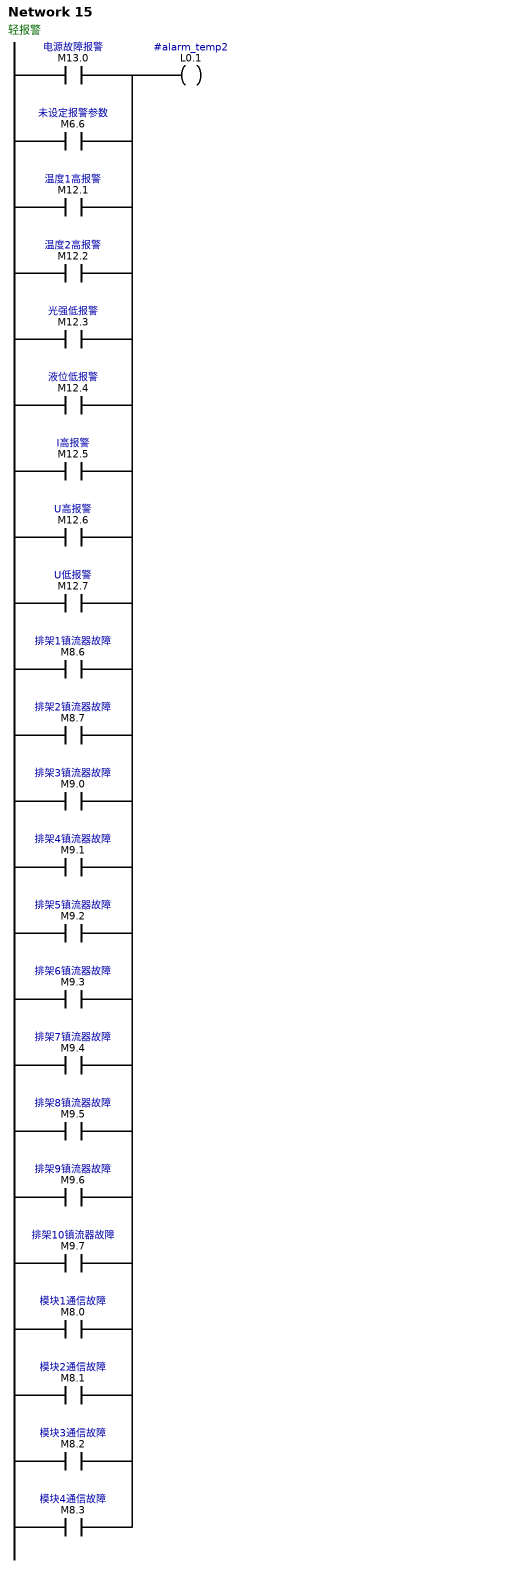
[picture p24: SBR7 networks 15-15]
Network 15
// 轻报警
LD     电源故障报警:M13.0
O      未设定报警参数:M6.6
O      温度1高报警:M12.1
O      温度2高报警:M12.2
O      光强低报警:M12.3
O      液位低报警:M12.4
O      I高报警:M12.5
O      U高报警:M12.6
O      U低报警:M12.7
O      排架1镇流器故障:M8.6
O      排架2镇流器故障:M8.7
O      排架3镇流器故障:M9.0
O      排架4镇流器故障:M9.1
O      排架5镇流器故障:M9.2
O      排架6镇流器故障:M9.3
O      排架7镇流器故障:M9.4
O      排架8镇流器故障:M9.5
O      排架9镇流器故障:M9.6
O      排架10镇流器故障:M9.7
O      模块1通信故障:M8.0
O      模块2通信故障:M8.1
O      模块3通信故障:M8.2
O      模块4通信故障:M8.3
=      #alarm_temp2:L0.1
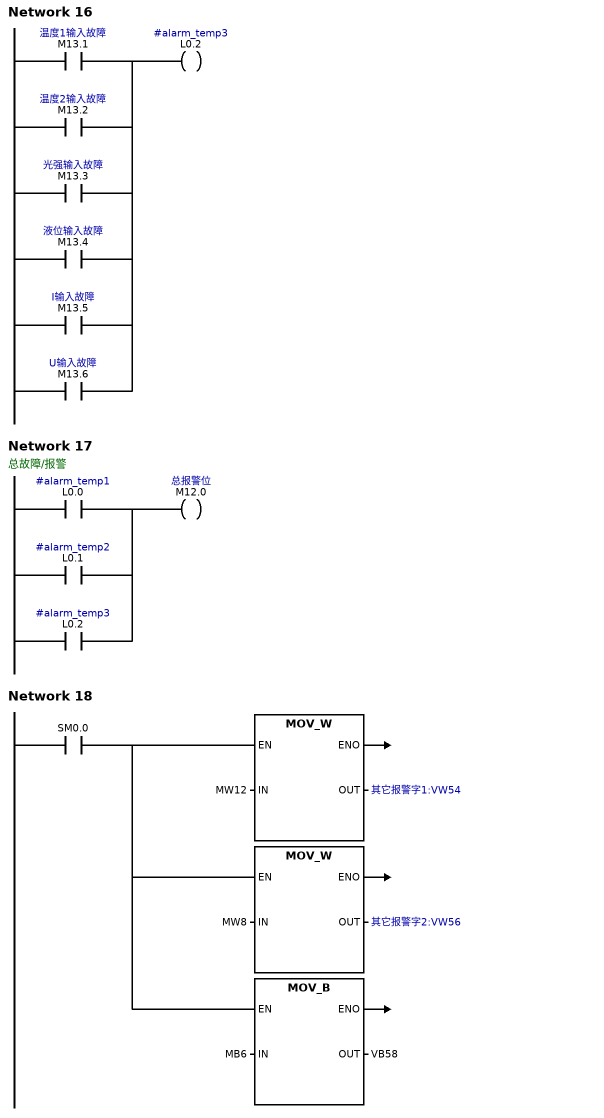
Network 16
LD     温度1输入故障:M13.1
O      温度2输入故障:M13.2
O      光强输入故障:M13.3
O      液位输入故障:M13.4
O      I输入故障:M13.5
O      U输入故障:M13.6
=      #alarm_temp3:L0.2
Network 17
// 总故障/报警
LD     #alarm_temp1:L0.0
O      #alarm_temp2:L0.1
O      #alarm_temp3:L0.2
=      总报警位:M12.0
Network 18
LD     SM0.0
MOVW   MW12, 其它报警字1:VW54
MOVW   MW8, 其它报警字2:VW56
MOVB   MB6, VB58
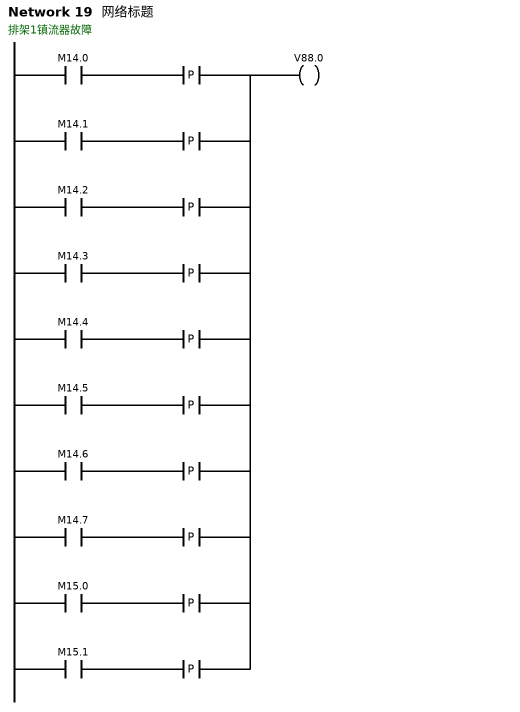
Network 19 // 网络标题
// 排架1镇流器故障
LD     M14.0
EU
LD     M14.1
EU
OLD
LD     M14.2
EU
OLD
LD     M14.3
EU
OLD
LD     M14.4
EU
OLD
LD     M14.5
EU
OLD
LD     M14.6
EU
OLD
LD     M14.7
EU
OLD
LD     M15.0
EU
OLD
LD     M15.1
EU
OLD
=      V88.0
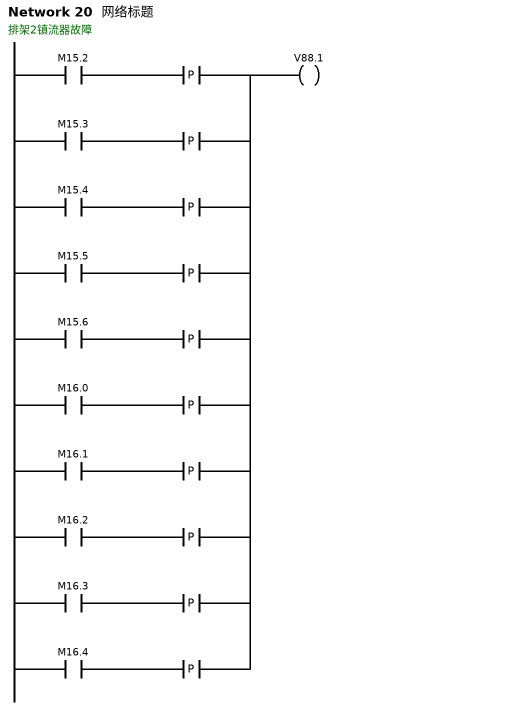
Network 20 // 网络标题
// 排架2镇流器故障
LD     M15.2
EU
LD     M15.3
EU
OLD
LD     M15.4
EU
OLD
LD     M15.5
EU
OLD
LD     M15.6
EU
OLD
LD     M16.0
EU
OLD
LD     M16.1
EU
OLD
LD     M16.2
EU
OLD
LD     M16.3
EU
OLD
LD     M16.4
EU
OLD
=      V88.1
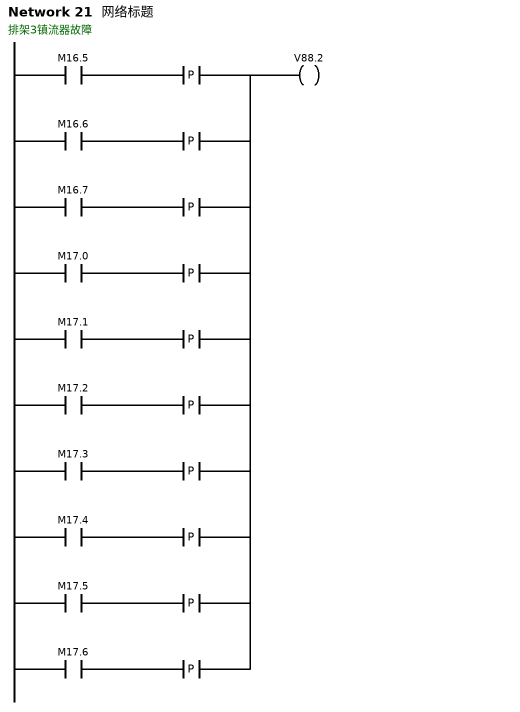
Network 21 // 网络标题
// 排架3镇流器故障
LD     M16.5
EU
LD     M16.6
EU
OLD
LD     M16.7
EU
OLD
LD     M17.0
EU
OLD
LD     M17.1
EU
OLD
LD     M17.2
EU
OLD
LD     M17.3
EU
OLD
LD     M17.4
EU
OLD
LD     M17.5
EU
OLD
LD     M17.6
EU
OLD
=      V88.2
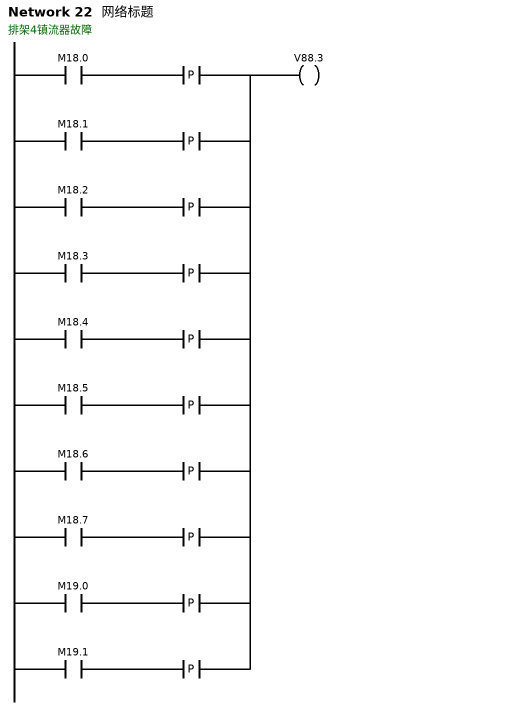
Network 22 // 网络标题
// 排架4镇流器故障
LD     M18.0
EU
LD     M18.1
EU
OLD
LD     M18.2
EU
OLD
LD     M18.3
EU
OLD
LD     M18.4
EU
OLD
LD     M18.5
EU
OLD
LD     M18.6
EU
OLD
LD     M18.7
EU
OLD
LD     M19.0
EU
OLD
LD     M19.1
EU
OLD
=      V88.3
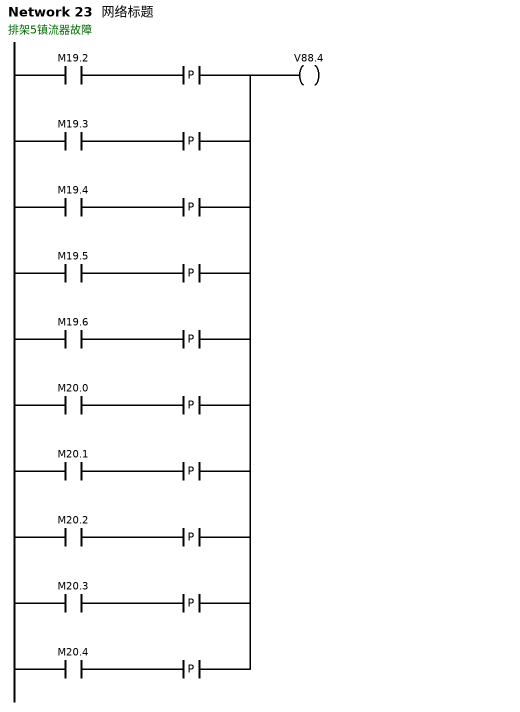
Network 23 // 网络标题
// 排架5镇流器故障
LD     M19.2
EU
LD     M19.3
EU
OLD
LD     M19.4
EU
OLD
LD     M19.5
EU
OLD
LD     M19.6
EU
OLD
LD     M20.0
EU
OLD
LD     M20.1
EU
OLD
LD     M20.2
EU
OLD
LD     M20.3
EU
OLD
LD     M20.4
EU
OLD
=      V88.4
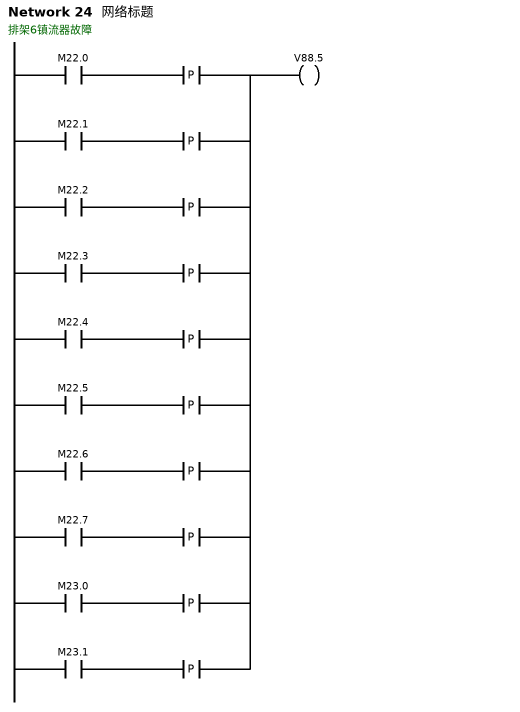
Network 24 // 网络标题
// 排架6镇流器故障
LD     M22.0
EU
LD     M22.1
EU
OLD
LD     M22.2
EU
OLD
LD     M22.3
EU
OLD
LD     M22.4
EU
OLD
LD     M22.5
EU
OLD
LD     M22.6
EU
OLD
LD     M22.7
EU
OLD
LD     M23.0
EU
OLD
LD     M23.1
EU
OLD
=      V88.5
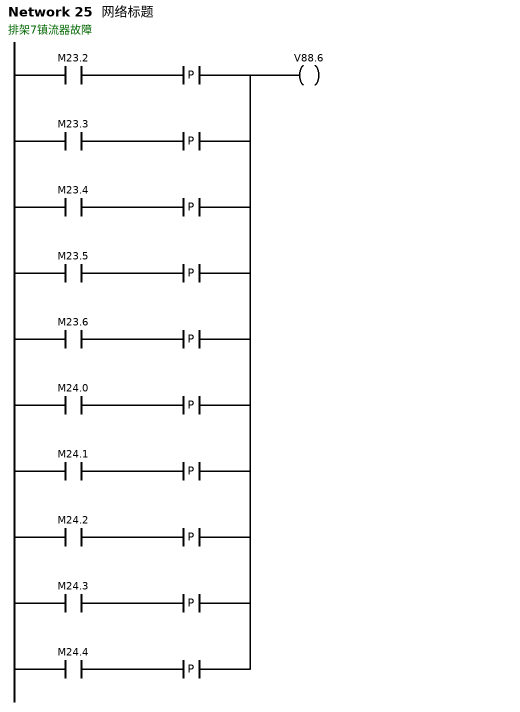
Network 25 // 网络标题
// 排架7镇流器故障
LD     M23.2
EU
LD     M23.3
EU
OLD
LD     M23.4
EU
OLD
LD     M23.5
EU
OLD
LD     M23.6
EU
OLD
LD     M24.0
EU
OLD
LD     M24.1
EU
OLD
LD     M24.2
EU
OLD
LD     M24.3
EU
OLD
LD     M24.4
EU
OLD
=      V88.6
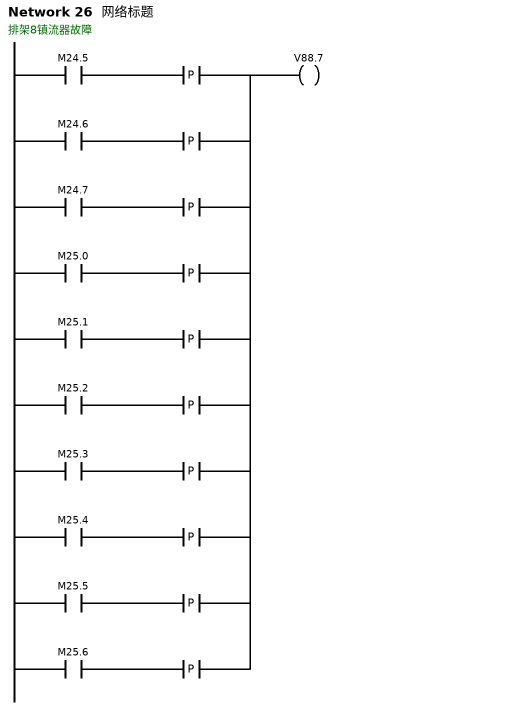
Network 26 // 网络标题
// 排架8镇流器故障
LD     M24.5
EU
LD     M24.6
EU
OLD
LD     M24.7
EU
OLD
LD     M25.0
EU
OLD
LD     M25.1
EU
OLD
LD     M25.2
EU
OLD
LD     M25.3
EU
OLD
LD     M25.4
EU
OLD
LD     M25.5
EU
OLD
LD     M25.6
EU
OLD
=      V88.7
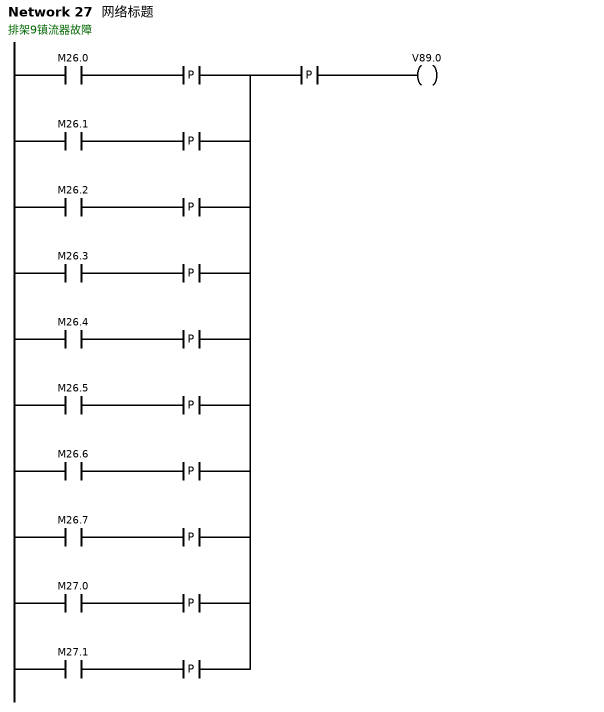
Network 27 // 网络标题
// 排架9镇流器故障
LD     M26.0
EU
LD     M26.1
EU
OLD
LD     M26.2
EU
OLD
LD     M26.3
EU
OLD
LD     M26.4
EU
OLD
LD     M26.5
EU
OLD
LD     M26.6
EU
OLD
LD     M26.7
EU
OLD
LD     M27.0
EU
OLD
LD     M27.1
EU
OLD
EU
=      V89.0
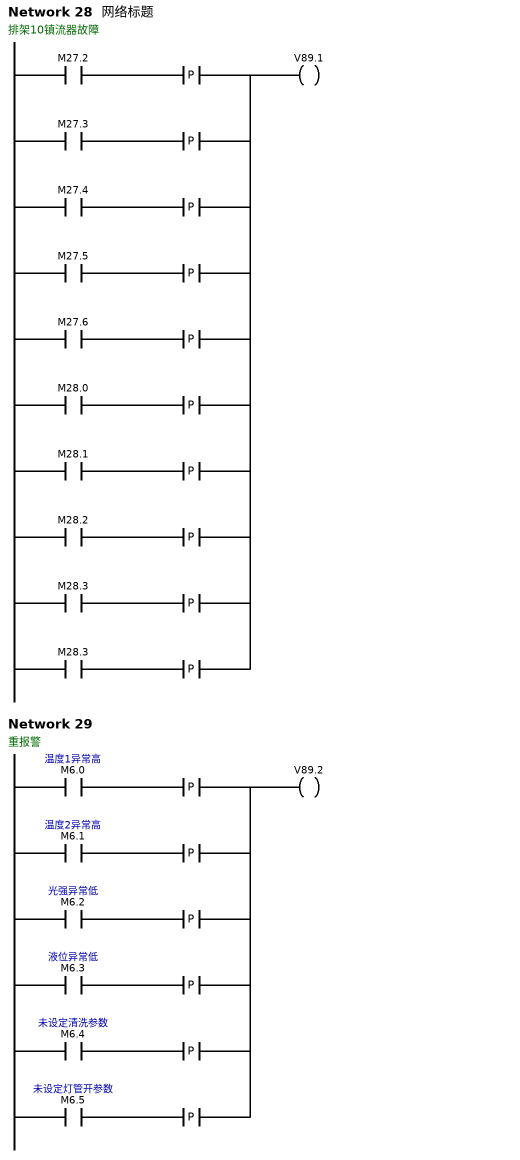
Network 28 // 网络标题
// 排架10镇流器故障
LD     M27.2
EU
LD     M27.3
EU
OLD
LD     M27.4
EU
OLD
LD     M27.5
EU
OLD
LD     M27.6
EU
OLD
LD     M28.0
EU
OLD
LD     M28.1
EU
OLD
LD     M28.2
EU
OLD
LD     M28.3
EU
OLD
LD     M28.3
EU
OLD
=      V89.1
Network 29
// 重报警
LD     温度1异常高:M6.0
EU
LD     温度2异常高:M6.1
EU
OLD
LD     光强异常低:M6.2
EU
OLD
LD     液位异常低:M6.3
EU
OLD
LD     未设定清洗参数:M6.4
EU
OLD
LD     未设定灯管开参数:M6.5
EU
OLD
=      V89.2
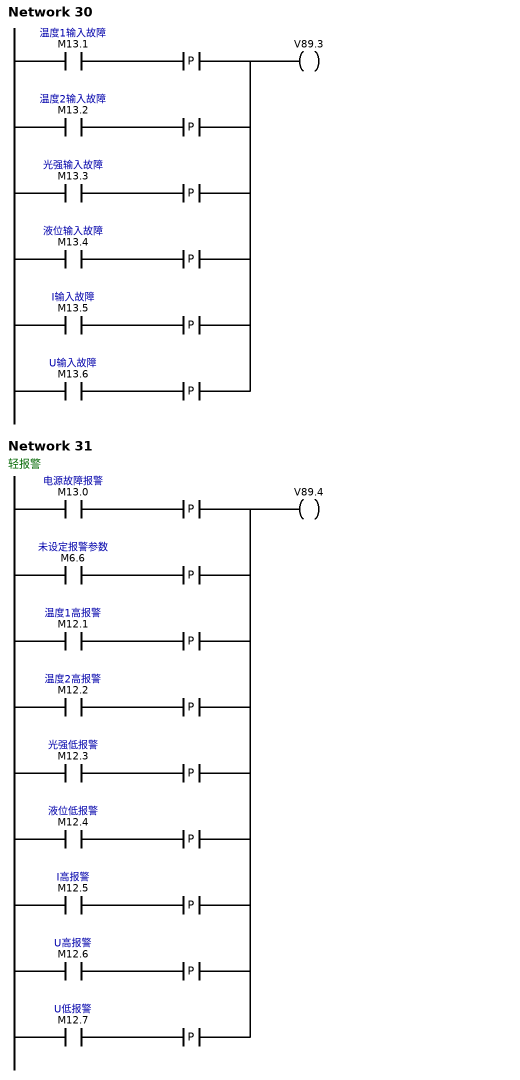
Network 30
LD     温度1输入故障:M13.1
EU
LD     温度2输入故障:M13.2
EU
OLD
LD     光强输入故障:M13.3
EU
OLD
LD     液位输入故障:M13.4
EU
OLD
LD     I输入故障:M13.5
EU
OLD
LD     U输入故障:M13.6
EU
OLD
=      V89.3
Network 31
// 轻报警
LD     电源故障报警:M13.0
EU
LD     未设定报警参数:M6.6
EU
OLD
LD     温度1高报警:M12.1
EU
OLD
LD     温度2高报警:M12.2
EU
OLD
LD     光强低报警:M12.3
EU
OLD
LD     液位低报警:M12.4
EU
OLD
LD     I高报警:M12.5
EU
OLD
LD     U高报警:M12.6
EU
OLD
LD     U低报警:M12.7
EU
OLD
=      V89.4
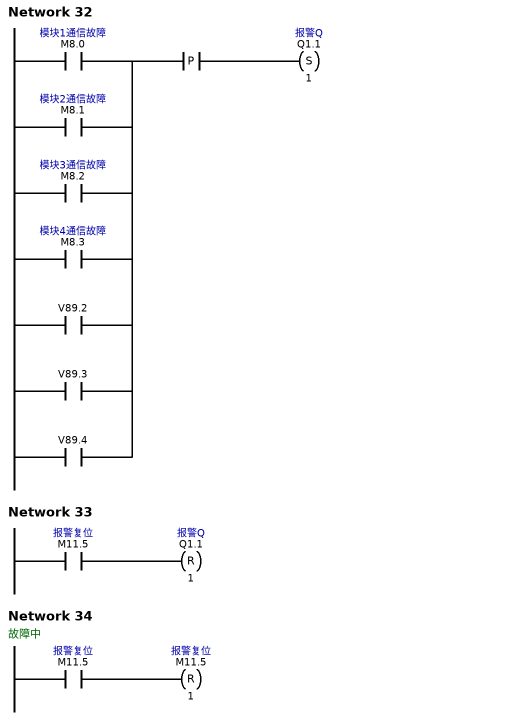
Network 32
LD     模块1通信故障:M8.0
O      模块2通信故障:M8.1
O      模块3通信故障:M8.2
O      模块4通信故障:M8.3
O      V89.2
O      V89.3
O      V89.4
EU
S      报警Q:Q1.1, 1
Network 33
LD     报警复位:M11.5
R      报警Q:Q1.1, 1
Network 34
// 故障中
LD     报警复位:M11.5
R      报警复位:M11.5, 1
END_SUBROUTINE_BLOCK

SUBROUTINE_BLOCK AD_INPUT:SBR8
TITLE=模拟量,单极性_0-32000,双极性:-32000-32000
//  将6个点划分为温度1,温度2,光强,水位,电压,电流,输入信号转化后与设置范围比较,得出最终真实值.
// 
VAR
Q:REAL;	// LD0 
END_VAR
BEGIN
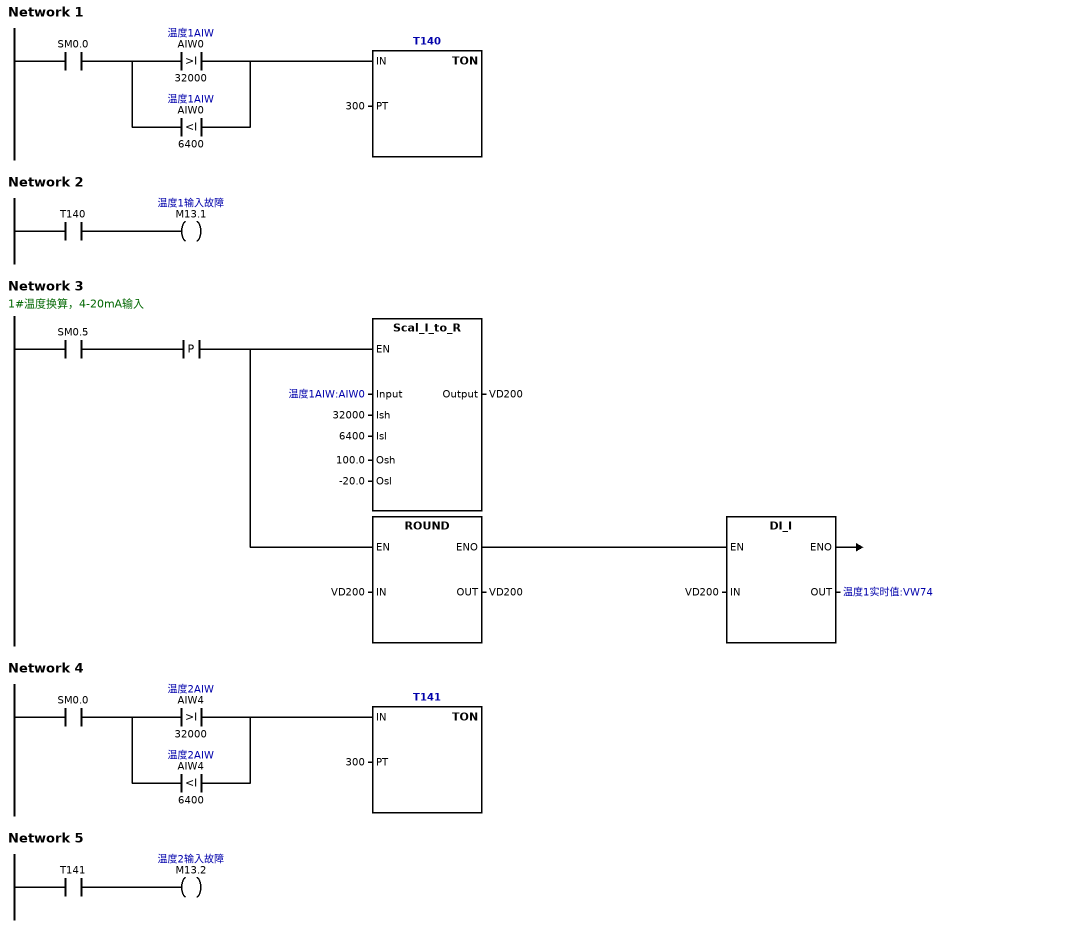
Network 1
LD     SM0.0
LDW>   温度1AIW:AIW0, 32000
OW<    温度1AIW:AIW0, 6400
ALD
TON    T140, 300
Network 2
LD     T140
=      温度1输入故障:M13.1
Network 3
// 1#温度换算，4-20mA输入
LD     SM0.5
EU
CALL   Scal_I_to_R:SBR9, 温度1AIW:AIW0, 32000, 6400, 100.0, -20.0, VD200
ROUND  VD200, VD200
AENO
DTI    VD200, 温度1实时值:VW74
Network 4
LD     SM0.0
LDW>   温度2AIW:AIW4, 32000
OW<    温度2AIW:AIW4, 6400
ALD
TON    T141, 300
Network 5
LD     T141
=      温度2输入故障:M13.2
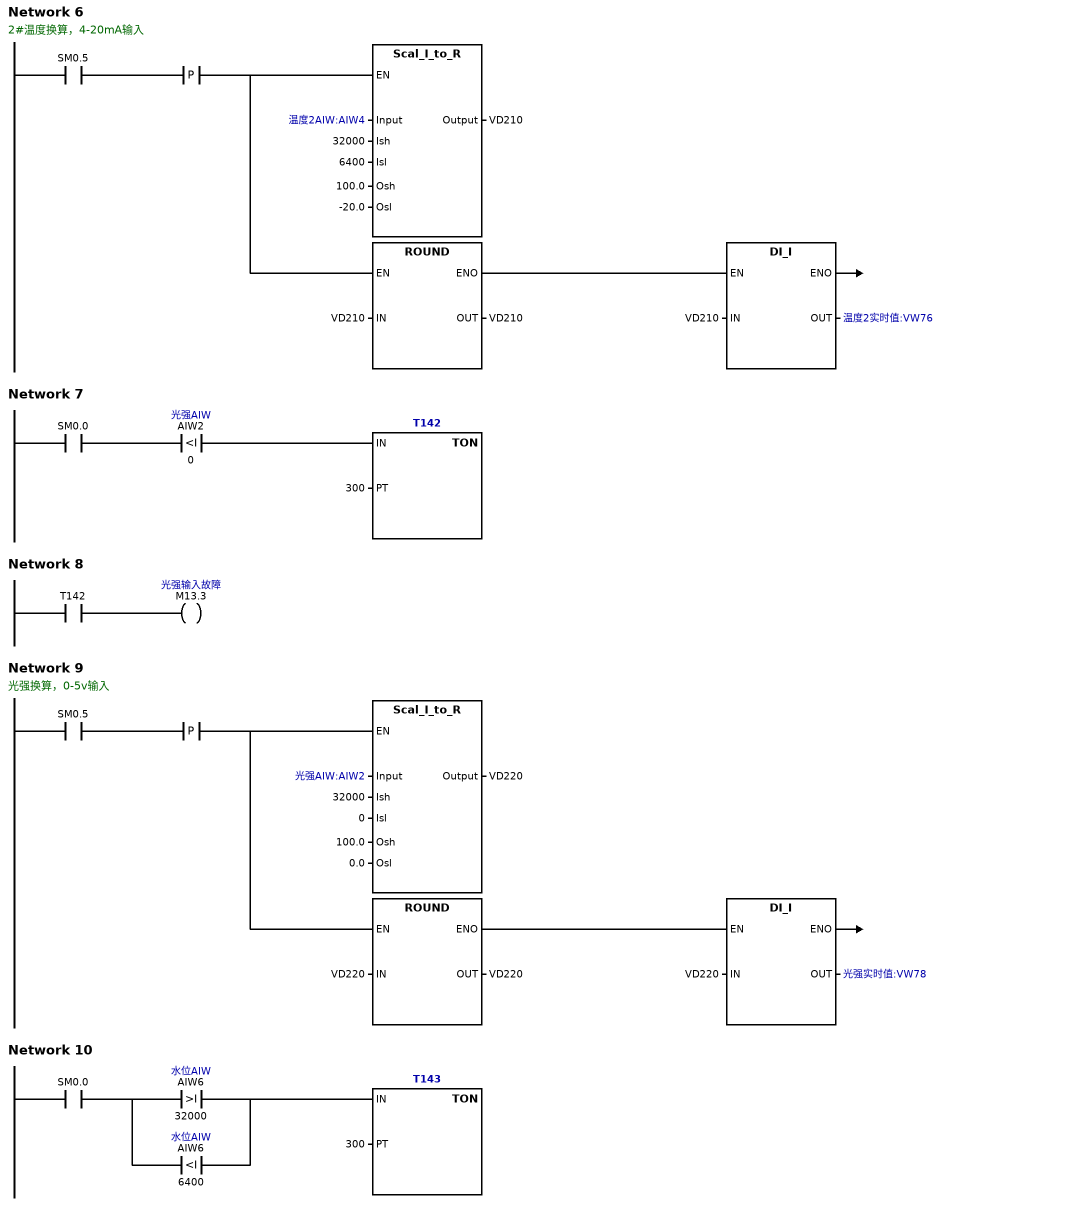
Network 6
// 2#温度换算，4-20mA输入
LD     SM0.5
EU
CALL   Scal_I_to_R:SBR9, 温度2AIW:AIW4, 32000, 6400, 100.0, -20.0, VD210
ROUND  VD210, VD210
AENO
DTI    VD210, 温度2实时值:VW76
Network 7
LD     SM0.0
AW<    光强AIW:AIW2, 0
TON    T142, 300
Network 8
LD     T142
=      光强输入故障:M13.3
Network 9
// 光强换算，0-5v输入
LD     SM0.5
EU
CALL   Scal_I_to_R:SBR9, 光强AIW:AIW2, 32000, 0, 100.0, 0.0, VD220
ROUND  VD220, VD220
AENO
DTI    VD220, 光强实时值:VW78
Network 10
LD     SM0.0
LDW>   水位AIW:AIW6, 32000
OW<    水位AIW:AIW6, 6400
ALD
TON    T143, 300
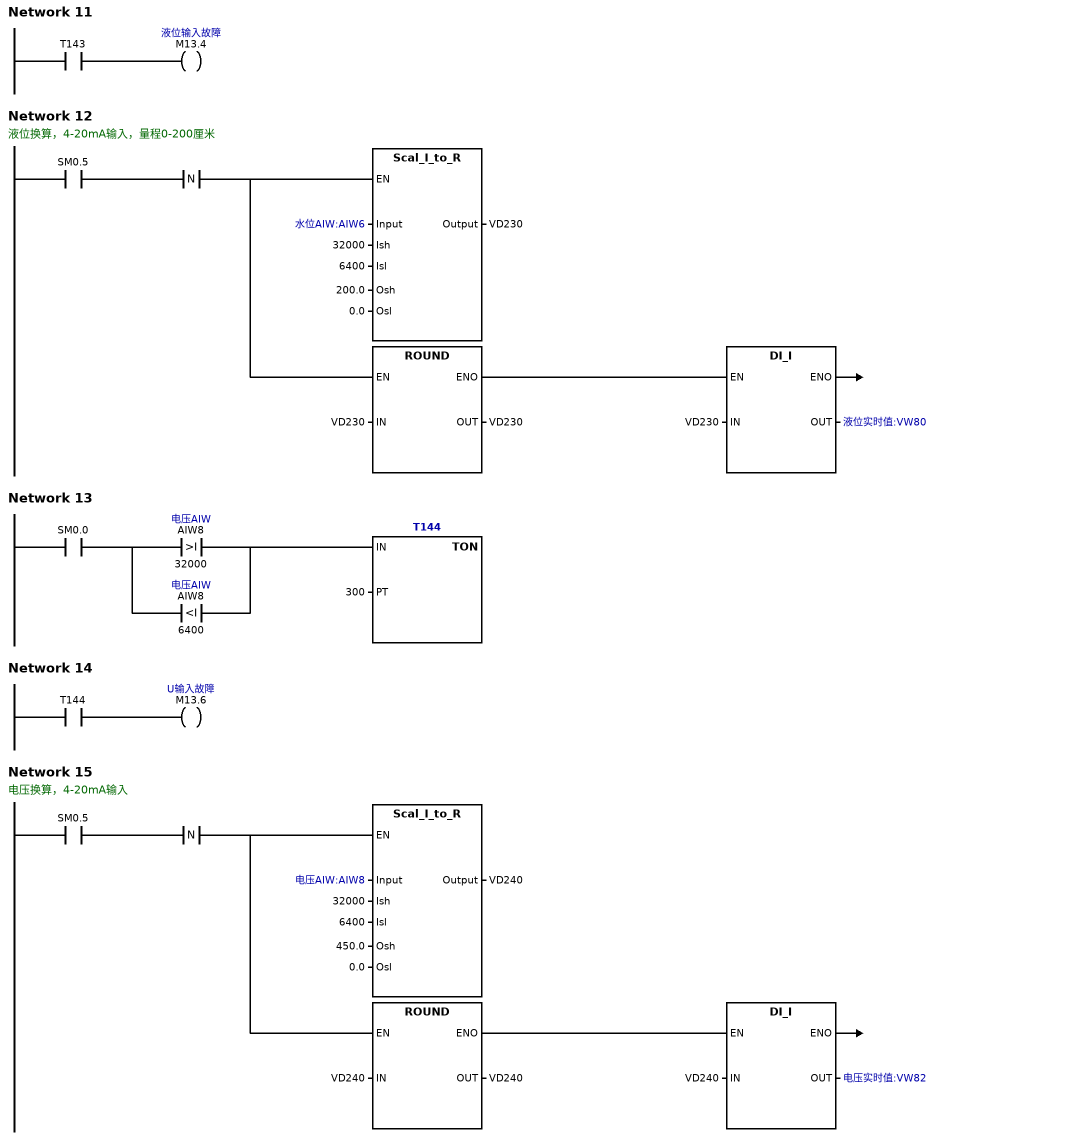
Network 11
LD     T143
=      液位输入故障:M13.4
Network 12
// 液位换算，4-20mA输入，量程0-200厘米
LD     SM0.5
ED
CALL   Scal_I_to_R:SBR9, 水位AIW:AIW6, 32000, 6400, 200.0, 0.0, VD230
ROUND  VD230, VD230
AENO
DTI    VD230, 液位实时值:VW80
Network 13
LD     SM0.0
LDW>   电压AIW:AIW8, 32000
OW<    电压AIW:AIW8, 6400
ALD
TON    T144, 300
Network 14
LD     T144
=      U输入故障:M13.6
Network 15
// 电压换算，4-20mA输入
LD     SM0.5
ED
CALL   Scal_I_to_R:SBR9, 电压AIW:AIW8, 32000, 6400, 450.0, 0.0, VD240
ROUND  VD240, VD240
AENO
DTI    VD240, 电压实时值:VW82
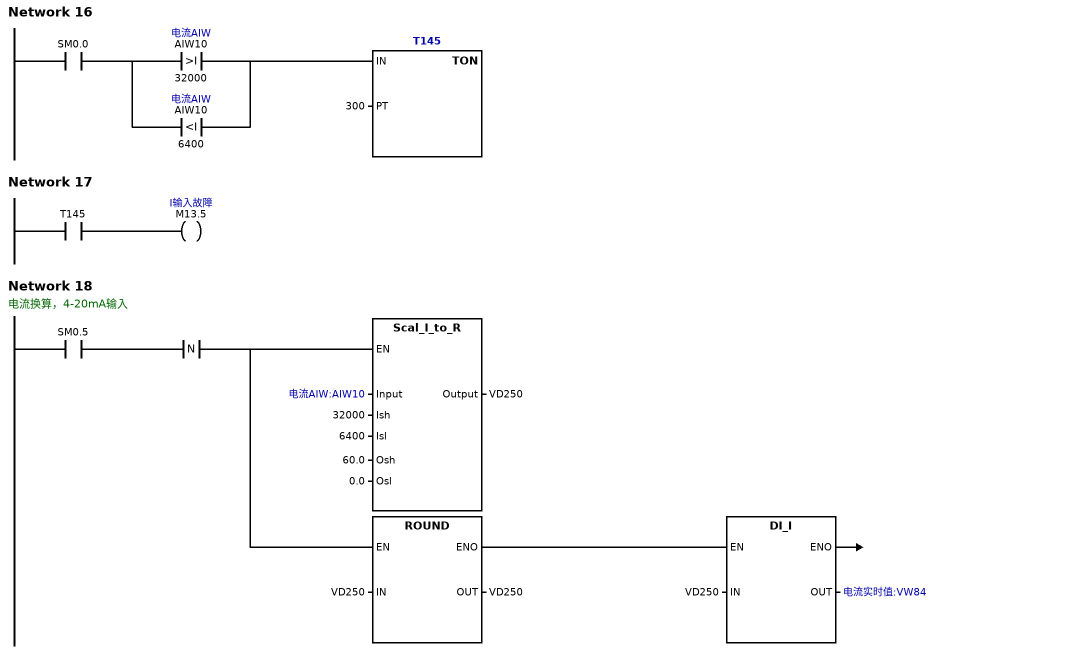
Network 16
LD     SM0.0
LDW>   电流AIW:AIW10, 32000
OW<    电流AIW:AIW10, 6400
ALD
TON    T145, 300
Network 17
LD     T145
=      I输入故障:M13.5
Network 18
// 电流换算，4-20mA输入
LD     SM0.5
ED
CALL   Scal_I_to_R:SBR9, 电流AIW:AIW10, 32000, 6400, 60.0, 0.0, VD250
ROUND  VD250, VD250
AENO
DTI    VD250, 电流实时值:VW84
END_SUBROUTINE_BLOCK

SUBROUTINE_BLOCK Scal_I_to_R:SBR9
TITLE=子程序注释
VAR_INPUT
Input:INT;	// LW0 
Ish:INT;	// LW2 
Isl:INT;	// LW4 
Osh:REAL;	// LD6 
Osl:REAL;	// LD10 
END_VAR
VAR_OUTPUT
Output:REAL;	// LD14 
END_VAR
VAR
Temp_D:DWORD;	// LD18 
Temp_R:REAL;	// LD22 
END_VAR
BEGIN
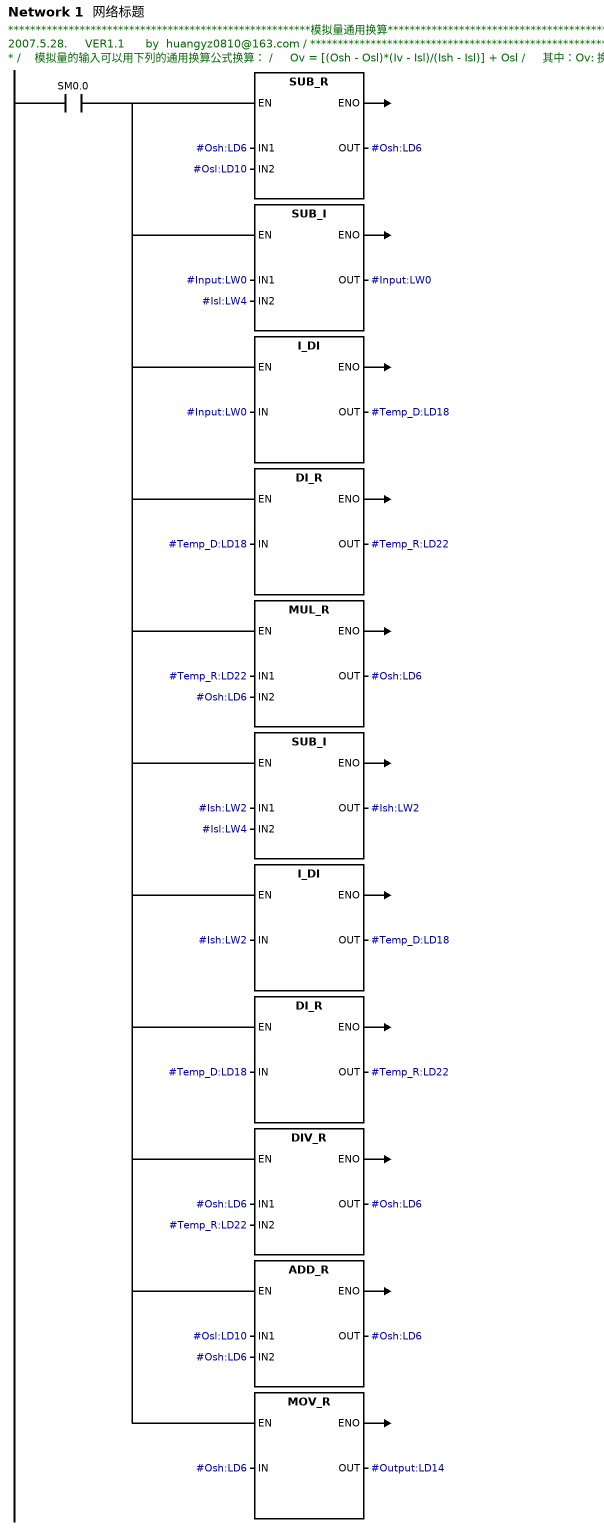
Network 1 // 网络标题
// *******************************************************模拟量通用换算**********************************************************************
// 2007.5.27.     VER1.0      by  huangyz0810@163.com     
// 2007.5.28.     VER1.1      by  huangyz0810@163.com
// **************************************************************************************************************************************************
//    模拟量的输入可以用下列的通用换算公式换算：
//     Ov = [(Osh - Osl)*(Iv - Isl)/(Ish - Isl)] + Osl
//     其中：Ov: 换算结果     Iv: 换算对象  Osl: 换算结果的低限
//     Ish: 换算对象的高限   Isl: 换算对象的低限
// 
// 
// (network saved uncompiled; LAD cells follow)
// row 0: c0 -| |- SM0.0 v  c1 --  c2 [SUB_R EN:=power@row0, IN1:=#Osh:LD6, IN2:=#Osl:LD10, ENO=>power, OUT=>#Osh:LD6]  c3 ->
// row 1: c0 ^v  c2 [box]
// row 2: c0 ^v  c1 --  c2 [SUB_I EN:=power@row2, IN1:=#Input:LW0, IN2:=#Isl:LW4, ENO=>power, OUT=>#Input:LW0]  c3 ->
// row 3: c0 ^v  c2 [box]
// row 4: c0 ^v  c1 --  c2 [I_DI EN:=power@row4, IN:=#Input:LW0, ENO=>power, OUT=>#Temp_D:LD18]  c3 ->
// row 5: c0 ^v  c2 [box]
// row 6: c0 ^v  c1 --  c2 [DI_R EN:=power@row6, IN:=#Temp_D:LD18, ENO=>power, OUT=>#Temp_R:LD22]  c3 ->
// row 7: c0 ^v  c2 [box]
// row 8: c0 ^v  c1 --  c2 [MUL_R EN:=power@row8, IN1:=#Temp_R:LD22, IN2:=#Osh:LD6, ENO=>power, OUT=>#Osh:LD6]  c3 ->
// row 9: c0 ^v  c2 [box]
// row 10: c0 ^v  c1 --  c2 [SUB_I EN:=power@row10, IN1:=#Ish:LW2, IN2:=#Isl:LW4, ENO=>power, OUT=>#Ish:LW2]  c3 ->
// row 11: c0 ^v  c2 [box]
// row 12: c0 ^v  c1 --  c2 [I_DI EN:=power@row12, IN:=#Ish:LW2, ENO=>power, OUT=>#Temp_D:LD18]  c3 ->
// row 13: c0 ^v  c2 [box]
// row 14: c0 ^v  c1 --  c2 [DI_R EN:=power@row14, IN:=#Temp_D:LD18, ENO=>power, OUT=>#Temp_R:LD22]  c3 ->
// row 15: c0 ^v  c2 [box]
// row 16: c0 ^v  c1 --  c2 [DIV_R EN:=power@row16, IN1:=#Osh:LD6, IN2:=#Temp_R:LD22, ENO=>power, OUT=>#Osh:LD6]  c3 ->
// row 17: c0 ^v  c2 [box]
// row 18: c0 ^v  c1 --  c2 [ADD_R EN:=power@row18, IN1:=#Osl:LD10, IN2:=#Osh:LD6, ENO=>power, OUT=>#Osh:LD6]  c3 ->
// row 19: c0 ^v  c2 [box]
// row 20: c0 ^  c1 --  c2 [MOV_R EN:=power@row20, IN:=#Osh:LD6, ENO=>power, OUT=>#Output:LD14]  c3 ->
// row 21: c2 [box]
END_SUBROUTINE_BLOCK

SUBROUTINE_BLOCK COMM_INIT:SBR50
TITLE=
BEGIN
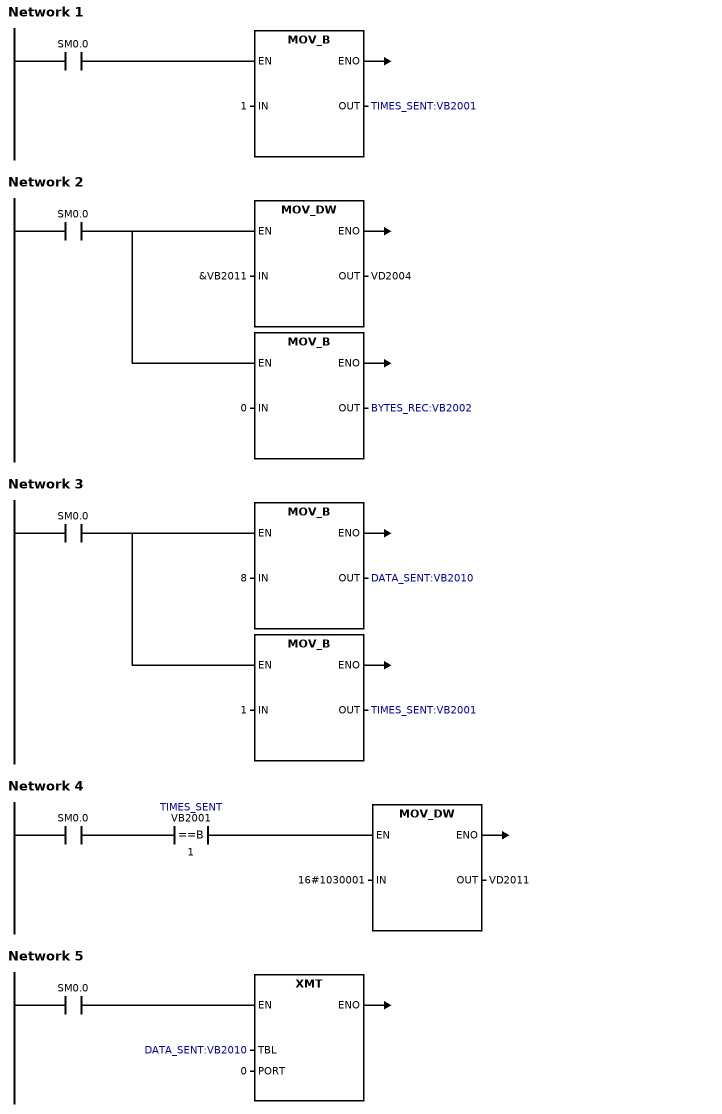
Network 1
LD     SM0.0
MOVB   1, TIMES_SENT:VB2001
Network 2
LD     SM0.0
MOVD   &VB2011, VD2004
MOVB   0, BYTES_REC:VB2002
Network 3
LD     SM0.0
MOVB   8, DATA_SENT:VB2010
MOVB   1, TIMES_SENT:VB2001
Network 4
LD     SM0.0
AB=    TIMES_SENT:VB2001, 1
MOVD   16#1030001, VD2011
Network 5
LD     SM0.0
XMT    DATA_SENT:VB2010, 0
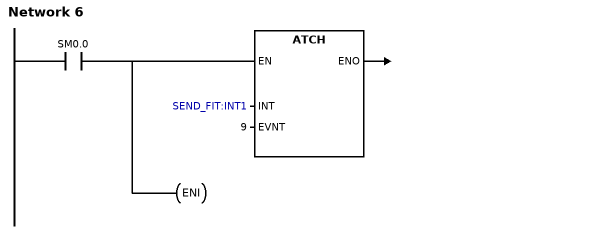
Network 6
LD     SM0.0
ATCH   SEND_FIT:INT1, 9
ENI
END_SUBROUTINE_BLOCK

SUBROUTINE_BLOCK COMM_CRC:SBR51
TITLE=
VAR_INPUT
COM_LEN:WORD;	// LW0 
CRC_PTR:DWORD;	// LD2 
END_VAR
VAR_OUTPUT
CRC:WORD;	// LW6 
END_VAR
BEGIN
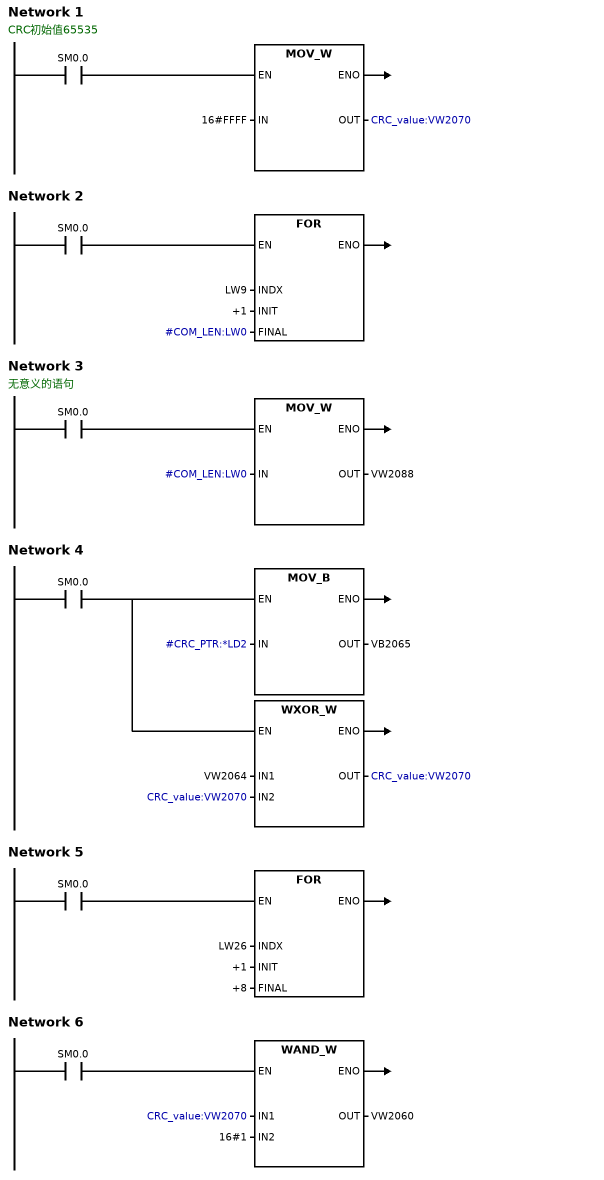
Network 1
// CRC初始值65535
// (network saved uncompiled; LAD cells follow)
// row 0: c0 -| |- SM0.0  c1 --  c2 [MOV_W EN:=power@row0, IN:=16#FFFF, ENO=>power, OUT=>CRC_value:VW2070]  c3 ->
// row 1: c2 [box]
Network 2
// (network saved uncompiled; LAD cells follow)
// row 0: c0 -| |- SM0.0  c1 --  c2 [FOR EN:=power@row0, INDX:=LW9, INIT:=+1, FINAL:=#COM_LEN:LW0, ENO=>power]  c3 ->
// row 1: c2 [box]
Network 3
// 无意义的语句
// (network saved uncompiled; LAD cells follow)
// row 0: c0 -| |- SM0.0  c1 --  c2 [MOV_W EN:=power@row0, IN:=#COM_LEN:LW0, ENO=>power, OUT=>VW2088]  c3 ->
// row 1: c2 [box]
Network 4
// (network saved uncompiled; LAD cells follow)
// row 0: c0 -| |- SM0.0 v  c1 --  c2 [MOV_B EN:=power@row0, IN:=*#CRC_PTR:LD2, ENO=>power, OUT=>VB2065]  c3 ->
// row 1: c0 ^v  c2 [box]
// row 2: c0 ^  c1 --  c2 [WXOR_W EN:=power@row2, IN1:=VW2064, IN2:=CRC_value:VW2070, ENO=>power, OUT=>CRC_value:VW2070]  c3 ->
// row 3: c2 [box]
Network 5
// (network saved uncompiled; LAD cells follow)
// row 0: c0 -| |- SM0.0  c1 --  c2 [FOR EN:=power@row0, INDX:=LW26, INIT:=+1, FINAL:=+8, ENO=>power]  c3 ->
// row 1: c2 [box]
Network 6
// (network saved uncompiled; LAD cells follow)
// row 0: c0 -| |- SM0.0  c1 --  c2 [WAND_W EN:=power@row0, IN1:=CRC_value:VW2070, IN2:=16#1, ENO=>power, OUT=>VW2060]  c3 ->
// row 1: c2 [box]
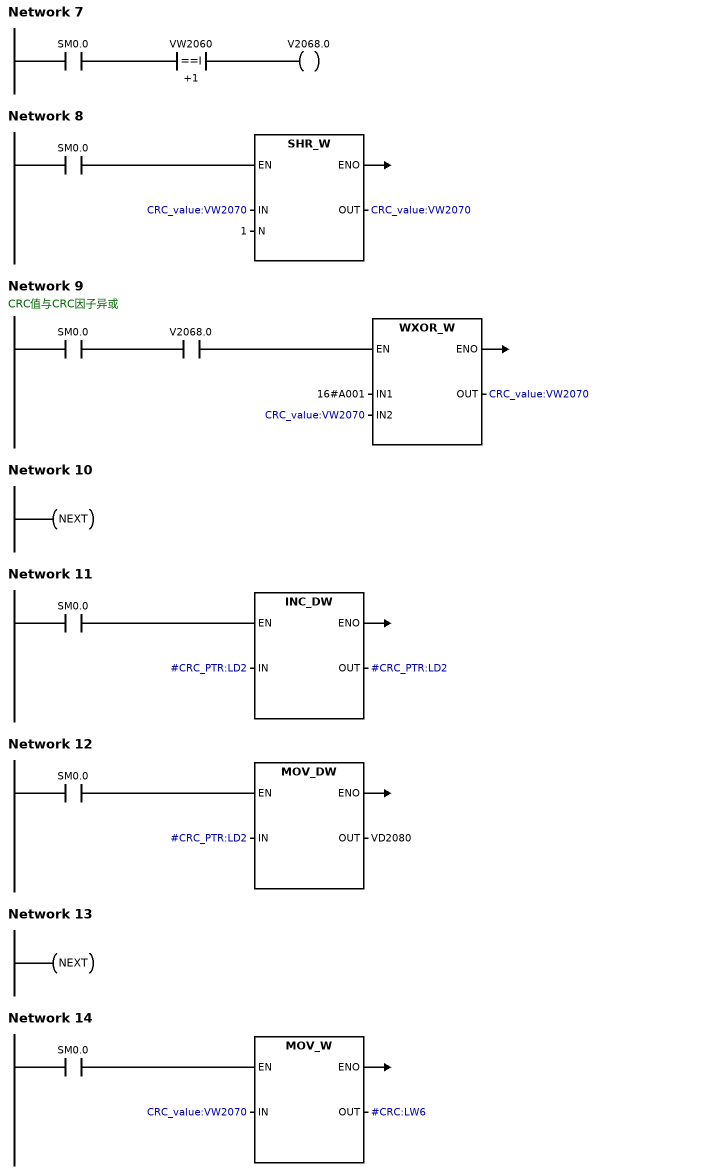
Network 7
// (network saved uncompiled; LAD cells follow)
// row 0: c0 -| |- SM0.0  c1 -|==I|- VW2060, +1  c2 -( ) V2068.0
Network 8
// (network saved uncompiled; LAD cells follow)
// row 0: c0 -| |- SM0.0  c1 --  c2 [SHR_W EN:=power@row0, IN:=CRC_value:VW2070, N:=1, ENO=>power, OUT=>CRC_value:VW2070]  c3 ->
// row 1: c2 [box]
Network 9
// CRC值与CRC因子异或
// (network saved uncompiled; LAD cells follow)
// row 0: c0 -| |- SM0.0  c1 -| |- V2068.0  c2 --  c3 [WXOR_W EN:=power@row0, IN1:=16#A001, IN2:=CRC_value:VW2070, ENO=>power, OUT=>CRC_value:VW2070]  c4 ->
// row 1: c3 [box]
Network 10
// (network saved uncompiled; LAD cells follow)
// row 0: c0 -(NEXT)
Network 11
// (network saved uncompiled; LAD cells follow)
// row 0: c0 -| |- SM0.0  c1 --  c2 [INC_DW EN:=power@row0, IN:=#CRC_PTR:LD2, ENO=>power, OUT=>#CRC_PTR:LD2]  c3 ->
// row 1: c2 [box]
Network 12
// (network saved uncompiled; LAD cells follow)
// row 0: c0 -| |- SM0.0  c1 --  c2 [MOV_DW EN:=power@row0, IN:=#CRC_PTR:LD2, ENO=>power, OUT=>VD2080]  c3 ->
// row 1: c2 [box]
Network 13
// (network saved uncompiled; LAD cells follow)
// row 0: c0 -(NEXT)
Network 14
// (network saved uncompiled; LAD cells follow)
// row 0: c0 -| |- SM0.0  c1 --  c2 [MOV_W EN:=power@row0, IN:=CRC_value:VW2070, ENO=>power, OUT=>#CRC:LW6]  c3 ->
// row 1: c2 [box]
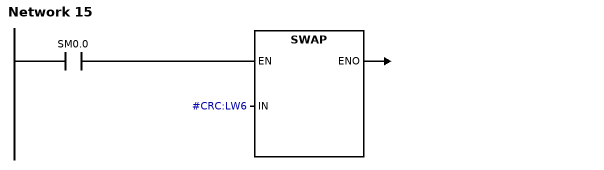
Network 15
// (network saved uncompiled; LAD cells follow)
// row 0: c0 -| |- SM0.0  c1 --  c2 [SWAP EN:=power@row0, IN:=#CRC:LW6, ENO=>power]  c3 ->
// row 1: c2 [box]
END_SUBROUTINE_BLOCK

SUBROUTINE_BLOCK DI_DATA:SBR52
TITLE=
BEGIN
